// Function block for AC motors controlled with the LENZE d-31855 frequency inverter
FUNCTION_BLOCK FB_Component_ACmotor IMPLEMENTS I_Component
VAR_INPUT
	// Interface vars
	sName			: STRING[20];
	bEnable     	: BOOL;
	//eMode       	: E_ComponentMode;
END_VAR

VAR_OUTPUT
	bE1jog1			: BOOL;					// jog func b1
	bE2jog2			: BOOL;					// jog func b2
	eE4Direction	: E_RotationDirection;	// motor direction
	// interface vars	
	eState			: E_ComponentState;
	iErrorCode		: INT;
	sStatusText 	: STRING[50];
END_VAR

VAR_IN_OUT
	bE3DCbrake		: BOOL;					// DC injection brake
END_VAR

VAR
	eJogFreq		: E_LenzeJogFreq;
END_VAR

IF bEnable AND eState = (E_ComponentState.READY OR E_ComponentState.BUSY) THEN
	// set jog frequency
	CASE eJogFreq OF
		E_LenzeJogFreq.F0HZ: 	bE1jog1 := FALSE;
								bE2jog2 := FALSE;
								eState	:= E_ComponentState.READY;
		E_LenzeJogFreq.F20HZ: 	bE1jog1 := TRUE;
								bE2jog2 := FALSE;
								eState	:= E_ComponentState.BUSY;
		E_LenzeJogFreq.F30HZ: 	bE1jog1 := FALSE;
								bE2jog2 := TRUE;
								eState	:= E_ComponentState.BUSY;
		E_LenzeJogFreq.F40HZ: 	bE1jog1 := TRUE;
								bE2jog2 := TRUE;
								eState	:= E_ComponentState.BUSY;
	END_CASE
	// DC braking
	IF bE3DCbrake THEN
		bE1jog1 := FALSE;
		bE2jog2 := FALSE;
		eState	:= E_ComponentState.BUSY;
	END_IF
ELSE
	bE1jog1 := FALSE;
	bE2jog2 := FALSE;
	eState	:= E_ComponentState.READY;
END_IF

{warning 'add method implementation '}
METHOD Halt : BOOL
bE1jog1 := FALSE;
bE2jog2 := FALSE;
eState := E_ComponentState.HALTED;
END_METHOD

METHOD SetDir : BOOL
VAR_INPUT
	Direction: E_RotationDirection;
END_VAR
eE4Direction := Direction;
END_METHOD

METHOD SetFreq : BOOL
VAR_INPUT
	Frequency: E_LenzeJogFreq;
END_VAR
eJogFreq := Frequency;
END_METHOD

{warning 'add method implementation '}
METHOD Start : BOOL
eState := E_ComponentState.READY;
END_METHOD

{warning 'add method implementation '}
METHOD Stop : BOOL
bE1jog1 := FALSE;
bE2jog2 := FALSE;
eState := E_ComponentState.DONE;
END_METHOD

END_FUNCTION_BLOCK

(* stored: Version 1.1.0.1, ProductVersion 3.1.4024.15
   POU FB_Component_ACmotor: Id {4bee0a47-7e8d-4a20-bf36-74643afc4427}, SpecialFunc None
   Method Halt: Id {86f47aa8-e6c4-4e8a-ae11-d7c42ced5250}
   Method SetDir: Id {d6a197ac-aaf3-4f2e-919c-b2334f169d78}
   Method SetFreq: Id {387ee47f-c4da-4cf1-a6b6-e28ea3f37257}
   Method Start: Id {8c2f0a58-166c-44b6-b1c3-800306693fc7}
   Method Stop: Id {84392872-6e4d-4fd5-a526-059b31207e24} *)
